FUNCTION_BLOCK AnalogStatus (* Composite Function Block Type *)
  (* Standard: 61499-2 *)
  (* Version 0.0, 7/3/2026, Schneider Electric, template *)
  PACKAGE SE.Nereda;
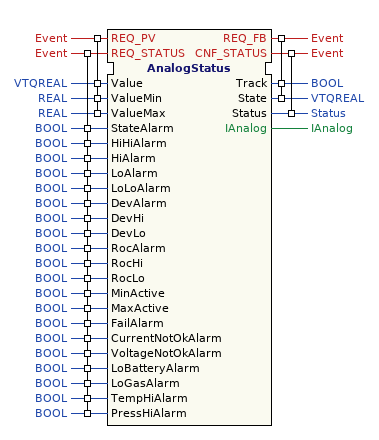
  EVENT_INPUT
    REQ_PV WITH Value, ValueMin, ValueMax; (* Request for new value and limits *)
    REQ_STATUS WITH HiHiAlarm, HiAlarm, LoAlarm, LoLoAlarm, DevAlarm, DevHi, DevLo, RocAlarm, RocHi, RocLo, MinActive, MaxActive, FailAlarm, CurrentNotOkAlarm, VoltageNotOkAlarm, LoBatteryAlarm, LoGasAlarm, TempHiAlarm, PressHiAlarm, StateAlarm; (* Execution request *)
  END_EVENT
  EVENT_OUTPUT
    REQ_FB WITH Track, State; (* Request for update of state and track *)
    CNF_STATUS WITH Status; (* Execution confirmation *)
  END_EVENT
  VAR_INPUT
    Value : VTQREAL; (* Vtq value *)
    ValueMin : REAL; (* Low limit of value *)
    ValueMax : REAL; (* High limit of value *)
    StateAlarm : BOOL; (* 1 = Alarm active *)
    HiHiAlarm : BOOL; (* 1 = High high alarm active *)
    HiAlarm : BOOL; (* 1 = High alarm active *)
    LoAlarm : BOOL; (* 1 = Low alarm active *)
    LoLoAlarm : BOOL; (* 1 = Low low alarm active *)
    DevAlarm : BOOL; (* 1 = Deviation alarm active, includes high and low deviation *)
    DevHi : BOOL; (* 1 = Deviation high active *)
    DevLo : BOOL; (* 1 = Devication low active *)
    RocAlarm : BOOL; (* 1 = Rate of change alarm active, includes high and low rate of change *)
    RocHi : BOOL; (* 1 = Rate of change high alarm active *)
    RocLo : BOOL; (* 1 = Rate of change low alarm active *)
    MinActive : BOOL; (* 1 = Value reached at minimum level *)
    MaxActive : BOOL; (* 1 = Value reached at  maximum level *)
    FailAlarm : BOOL; (* 1 = Fail alarm from the device is active *)
    CurrentNotOkAlarm : BOOL; (* 1 = Current value from field is not ok *)
    VoltageNotOkAlarm : BOOL; (* 1 = Voltage value from field is not ok *)
    LoBatteryAlarm : BOOL; (* 1 = Low battery alarm is active *)
    LoGasAlarm : BOOL; (* 1 = Low gas alarm is active *)
    TempHiAlarm : BOOL; (* 1 = Temperature high alarm is active *)
    PressHiAlarm : BOOL; (* 1 = Pressure high alarm is active *)
  END_VAR
  VAR_OUTPUT
    Track : BOOL; (* Tracking setpoint *)
    State : VTQREAL; (* Current state *)
    Status : Status; (* Status structure data (State alarm, HiHi alarm, Hi alarm, Lo alarm, LoLo alarm, Deviation alarm, Deviation Hi, Deivation Lo, ROC alarm, ROC Hi, ROC Lo, Min activated, Max activated) *)
  END_VAR
  PLUGS
    IAnalog : IAnalog;
  END_PLUGS
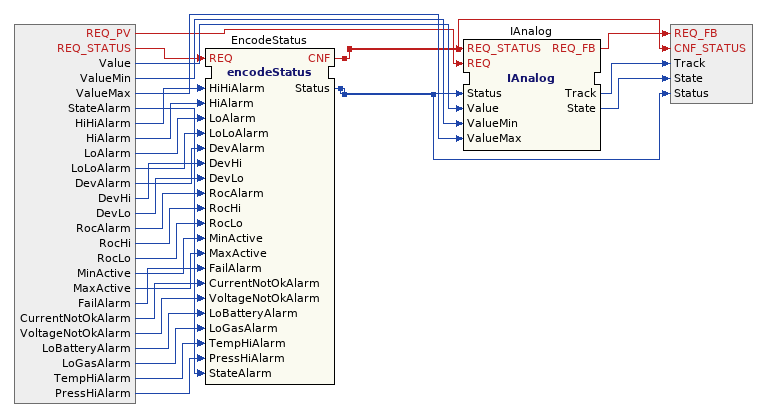
  FBS
    EncodeStatus : encodeStatus;
  END_FBS
  EVENT_CONNECTIONS
    EncodeStatus.CNF TO IAnalog.REQ_STATUS;
    REQ_PV TO IAnalog.REQ;
    REQ_STATUS TO EncodeStatus.REQ;
    IAnalog.REQ_FB TO REQ_FB;
    EncodeStatus.CNF TO CNF_STATUS;
  END_CONNECTIONS
  DATA_CONNECTIONS
    EncodeStatus.Status TO IAnalog.Status;
    Value TO IAnalog.Value;
    ValueMin TO IAnalog.ValueMin;
    ValueMax TO IAnalog.ValueMax;
    HiHiAlarm TO EncodeStatus.HiHiAlarm;
    HiAlarm TO EncodeStatus.HiAlarm;
    LoAlarm TO EncodeStatus.LoAlarm;
    LoLoAlarm TO EncodeStatus.LoLoAlarm;
    DevAlarm TO EncodeStatus.DevAlarm;
    DevHi TO EncodeStatus.DevHi;
    DevLo TO EncodeStatus.DevLo;
    RocAlarm TO EncodeStatus.RocAlarm;
    RocHi TO EncodeStatus.RocHi;
    RocLo TO EncodeStatus.RocLo;
    MinActive TO EncodeStatus.MinActive;
    MaxActive TO EncodeStatus.MaxActive;
    FailAlarm TO EncodeStatus.FailAlarm;
    CurrentNotOkAlarm TO EncodeStatus.CurrentNotOkAlarm;
    VoltageNotOkAlarm TO EncodeStatus.VoltageNotOkAlarm;
    LoBatteryAlarm TO EncodeStatus.LoBatteryAlarm;
    LoGasAlarm TO EncodeStatus.LoGasAlarm;
    TempHiAlarm TO EncodeStatus.TempHiAlarm;
    PressHiAlarm TO EncodeStatus.PressHiAlarm;
    IAnalog.Track TO Track;
    IAnalog.State TO State;
    StateAlarm TO EncodeStatus.StateAlarm;
    EncodeStatus.Status TO Status;
  END_CONNECTIONS
END_FUNCTION_BLOCK
